TYPE S_POSITION2D :
STRUCT
	X : LREAL;
	Y : LREAL;
END_STRUCT
END_TYPE

(* stored: Version 1.1.0.1, ProductVersion 3.1.4019.2
   DUT S_POSITION2D: Id {d2b5b6e6-aaa7-4b67-a4cb-3dbcfb182011} *)
